FUNCTION_BLOCK FB_AutoStartPos
VAR_INPUT
	bEnable 						: BOOL; 
	fPosition						: LREAL;
	fStartPosition					: LREAL;
	
	eStatus 						: BOOL; //E_Status;
	bAutoSineOff					: BOOL;
END_VAR
VAR_OUTPUT
	bStartPosOK						: BOOL;
	fWinchValveNormalizedInput 		: LREAL;
	bOpenBreak						: BOOL;
END_VAR

VAR PERSISTENT
	fProportionalGain 				: LREAL;
	fIntegralGain					: LREAL;
	fDerivateGain					: LREAL;
END_VAR

VAR
	fbPID_controller				: FB_PID_controller;
	fPosition_error					: LREAL;
	fProportinalGain_output			: LREAL;
	fIntegralGain_output			: LREAL;
	fDerivateGain_output			: LREAL;
	bEnableValveOutputWinch			: BOOL;	
	
	//Soft Start
	u								: LREAL;
	y								: LREAL;
	fTotal_distance					: LREAL;
	bAutoSineOff_prev				: BOOL;
END_VAR

IF eStatus AND G_Engineer_HMI.bAutoStartPosEnable THEN
	bOpenBreak	:= TRUE;
ELSE
	bOpenBreak := FALSE;
END_IF

IF bEnable  THEN
fPosition_error := fStartPosition - fPosition; //fPosition - fStartPosition;
G_Motion_Control.fPosition_error_StartPos := fPosition_error;


/////Soft Start//////

(*
IF NOT(bAutoSineOff) AND bAutoSineOff_prev THEN
fTotal_distance := ABS(fStartPosition - fPosition);
END_IF

bAutoSineOff_prev := bAutoSineOff;

u := fPosition_error/fTotal_distance;

IF u > 0.5 THEN
y := 1 - ((3*u*u) - (2*u*u*u)); 
END_IF

IF u < 0.5 THEN
	y := ((3*u*u) - (2*u*u*u)); 
END_IF

IF u < 0.0 THEN
	u := 0.0;
END_IF*)

// Write to HMI
//PGain:
IF NOT(G_Engineer_HMI.bPenable_MOOG_write) THEN
	G_Engineer_HMI.fProportionalgain_MOOG := fProportionalGain; // SKjønner ikke helt det her
ELSE
	fProportionalGain := G_Engineer_HMI.fProportionalgain_MOOG;
END_IF

//IGain: 
IF NOT(G_Engineer_HMI.bIenable_MOOG_write) THEN
	G_Engineer_HMI.fIntegrationalgain_MOOG := fIntegralGain;
ELSE
	fIntegralGain := G_Engineer_HMI.fIntegrationalgain_MOOG;
END_IF

fbPID_controller(
		ssMethodType := BOOL_TO_SINT(bEnable),
		error := fPosition_error,
		Int_error_threshold := G_PID_Tuning.Int_error_threshold,
		P_enable := G_Engineer_HMI.bPenable_MOOG,
		I_enable := G_Engineer_HMI.bIenable_MOOG,
		D_enable := FALSE,
		K_p := fProportionalGain,
		K_i := fIntegralGain,
		K_d := fDerivateGain,
		P_output => fProportinalGain_output,
		I_output => fIntegralGain_output,
		D_output => fDerivateGain_output
		);
		
			//Error times PGain
	fProportinalGain_output := fProportinalGain_output;
	G_PID_Tuning.fProportinalGain_output_MOOG := fProportinalGain_output;
	//Error times IGain
	fIntegralGain_output := fIntegralGain_output;
	G_PID_Tuning.fIntegralGain_output_MOOG := fIntegralGain_output;
	//Error times DGain
	fDerivateGain_output := fDerivateGain_output;
	G_PID_Tuning.fDerivateGain_output_MOOG := fDerivateGain_output;
	
	//Normalized Outputsignal
		
		fWinchValveNormalizedInput := LIMIT(-1, (fProportinalGain_output + fIntegralGain_output + fDerivateGain_output), 1); //Legg in y for å bruke soft start
		G_PID_Tuning.PID_output_MOOG := fWinchValveNormalizedInput;
		
	
	IF ABS(fPosition_error) < 0.05 THEN
		bStartPosOK := TRUE;
	END_IF
		
ELSE
	bStartPosOK := FALSE;
END_IF

END_FUNCTION_BLOCK

(* stored: Version 1.1.0.1
   POU FB_AutoStartPos: Id {bc9cc522-7b04-40cd-ac55-3a13b0903ef0}, SpecialFunc None *)
